FUNCTION_BLOCK Byte2DoubleArray (* Basic Function Block Type *)
  (* Standard: 61499-2 *)
  (* Version 0.0, 12/6/2015, gulzha, nxtControl GmbH, Template *)
  PACKAGE Main;
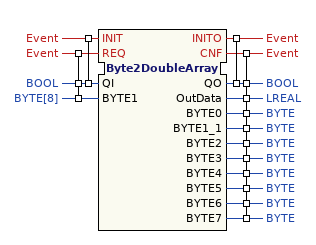
  EVENT_INPUT
    INIT WITH QI; (* Initialization Request *)
    REQ WITH QI, BYTE1; (* Normal Execution Request *)
  END_EVENT
  EVENT_OUTPUT
    INITO WITH QO; (* Initialization Confirm *)
    CNF WITH QO, OutData, BYTE0, BYTE1_1, BYTE2, BYTE3, BYTE4, BYTE5, BYTE6, BYTE7; (* Execution Confirmation *)
  END_EVENT
  VAR_INPUT
    QI : BOOL; (* Input event qualifier *)
    BYTE1 : ARRAY [0..7] OF BYTE;
  END_VAR
  VAR_OUTPUT
    QO : BOOL; (* Output event qualifier *)
    OutData : LREAL;
    BYTE0 : BYTE;
    BYTE1_1 : BYTE;
    BYTE2 : BYTE;
    BYTE3 : BYTE;
    BYTE4 : BYTE;
    BYTE5 : BYTE;
    BYTE6 : BYTE;
    BYTE7 : BYTE;
  END_VAR
  VAR
    temp : LWORD;
    i : INT;
    tempByte : BYTE;
  END_VAR
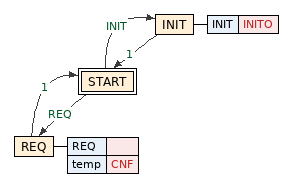
  EC_STATES
    START; (* Initial State *)
    INIT : INIT -> INITO; (* Initialization *)
    REQ : REQ, temp -> CNF; (* Normal execution *)
  END_STATES
  EC_TRANSITIONS
    START TO INIT := INIT;
    INIT TO START := 1;
    START TO REQ := REQ;
    REQ TO START := 1;
  END_TRANSITIONS
  ALGORITHM INIT IN ST: (* Initialization algorithm *)
;
  END_ALGORITHM
  ALGORITHM REQ IN ST: (* Normally executed algorithm *)
;

temp := 0;
//4bytesData := (SHL(SHL(SHL(BYTE_TO_DWORD(in1), 8) OR BYTE_TO_DWORD(in2), 8) OR     BYTE_TO_DWORD(in3), 8) OR in4);

//temp:= BYTE_TO_LREAL(Inputarray[0])
(*temp:= (SHL((temp OR BYTE1[0]),56) OR SHL((temp OR BYTE1[1]),48) OR
        SHL((temp OR BYTE1[2]),40) OR SHL((temp OR BYTE1[3]),32) OR
        SHL((temp OR BYTE1[4]),24) OR SHL((temp OR BYTE1[5]),16) OR
        SHL((temp OR BYTE1[6]),8) OR (temp OR BYTE1[7]));*)
temp := temp OR BYTE1[7];
temp:=  SHL(temp,8);
temp := temp OR BYTE1[6];
temp:=  SHL(temp,8);
temp := temp OR BYTE1[5];
temp:=  SHL(temp,8);
temp := temp OR BYTE1[4];
temp:=  SHL(temp,8);
temp := temp OR BYTE1[3];
temp:=  SHL(temp,8);
temp := temp OR BYTE1[2];
temp:=  SHL(temp,8);
temp := temp OR BYTE1[1];
temp:=  SHL(temp,8);
temp := temp OR BYTE1[0];

OutData:=DWORD_TO_LREAL(temp);
//OutData:= DWORD_TO_REAL(temp); //LREAL_TO_DWORD();
  END_ALGORITHM
  ALGORITHM temp IN ST:
;

BYTE0:=BYTE1[0];
BYTE1_1:=BYTE1[1];
BYTE2:=BYTE1[2];
BYTE3:=BYTE1[3];
BYTE4:=BYTE1[4];
BYTE5:=BYTE1[5];
BYTE6:=BYTE1[6];
BYTE7:=BYTE1[7];
  END_ALGORITHM
END_FUNCTION_BLOCK
